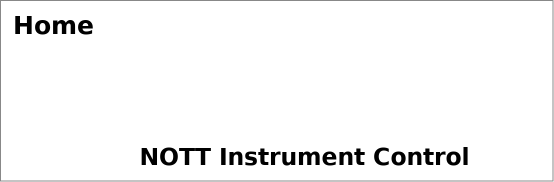
VISUALIZATION VISU_HMI_HOME  // 554x182
VAR_IN_OUT
	m_instance : FB_NOTT_ICS;
END_VAR
    Label (10,10 150x30), "Home"
    Label (56,132 498x50), "NOTT Instrument Control"
END_VISUALIZATION

(* stored: Version 1.1.0.1, ProductVersion 3.1.4024.14
   Visu VISU_HMI_HOME: Id {8b279cc1-e8ff-49da-81e2-69443df461ca} *)
